(* IEC 61131-3 sources: CodesysTest/alpha/export/Pro18_1174_04.dev/Plc Logic/Application/Motors/Applied Motion/FB_AppliedMotionBagDeliveryMotorNoFollowing.pou, 2 files *)

(* ---- FB_AppliedMotionBagDeliveryMotorNoFollowing.pou.st ---- *)
(*#-#-#-#-#-#-#-#-#-#---Declaration---#-#-#-#-#-#-#-#-#-#-#-#-#*)

FUNCTION_BLOCK FB_AppliedMotionBagDeliveryMotorNoFollowing EXTENDS FB_AppliedMotionStepServoEIPBase
VAR_INPUT
END_VAR
VAR_OUTPUT
END_VAR
VAR
	_moveDistance : BOOL;
	_moveDistanceONS : R_TRIG;
	_moveFinal : BOOL;
	_moveFinalONS : R_TRIG;
	_moveDone : BOOL;
	waitForMove : TON := (PT := T#30MS);
	manualFinalMovePB : BOOL;
	movedFinal : BOOL;
	moveDistanceState : BAG_DELIVERY_MOVE_STATES;
	moveDistanceFinalState : BAG_DELIVERY_MOVE_STATES;
END_VAR
(*#-#-#-#-#-#-#-#-#-#---Implementation---#-#-#-#-#-#-#-#-#-#-#-#-#*)

(* ---- MoveDistance.m.st ---- *)
(*#-#-#-#-#-#-#-#-#-#---Declaration---#-#-#-#-#-#-#-#-#-#-#-#-#*)

METHOD MoveDistance
VAR_INPUT
    distance : REAL;        //Distance to move in inches
    acceleration : INT;        //Acceleration in RPM/sec
    deceleration : INT;        //Deceleration in RPM/sec
    velocity : INT;            //Velocity in .25RPM
END_VAR(*#-#-#-#-#-#-#-#-#-#---Implementation---#-#-#-#-#-#-#-#-#-#-#-#-#*)

commandSuccessful := FALSE;
_moveDone := FALSE;
moveDistanceState := BAG_DELIVERY_MOVE_STATES.Idle;
distanceToMoveInSteps := REAL_TO_DINT((distance) * stepsPerInchSetpoint);

IF reversePolarity THEN
    distanceToMoveInSteps := distanceToMoveInSteps * -1;
END_IF

pointToPointAccelSetpoint := acceleration;
pointToPointDecelSetpoint := deceleration;
velocitySetpoint := velocity;

currentLimit := defaultCurrentSetpoint;
_moveDistance := TRUE;

//commands.feedToLength := TRUE;
//SUPER^.ExecuteStoredProgram(1);
